// TIA Portal V17 export
// export: Created 2024-06-25T12:57:18.7892853Z, ExportSetting WithDefaults, DisplayName Totally Integrated Automation Portal, DisplayVersion V17 Update 6, DisplayName TIA Portal Openness, DisplayVersion V17 Update 6, DisplayName TIA Portal Version Control Interface, DisplayVersion V17, DisplayName STEP 7 Professional, DisplayVersion V17 Update 6, DisplayName STEP 7 Safety, DisplayVersion V17 Update 6, DisplayName WinCC Advanced, DisplayVersion V17 Update 6
FUNCTION "Salidas" : Void   // FC5, LAD
{ S7_Optimized_Access := 'TRUE' }
VERSION : 0.1
// stored: AutoNumber true, IsIECCheckEnabled false, SetENOAutomatically false, UDAEnableTagReadback false
BEGIN

REGION Network 1: PILOTO OFF
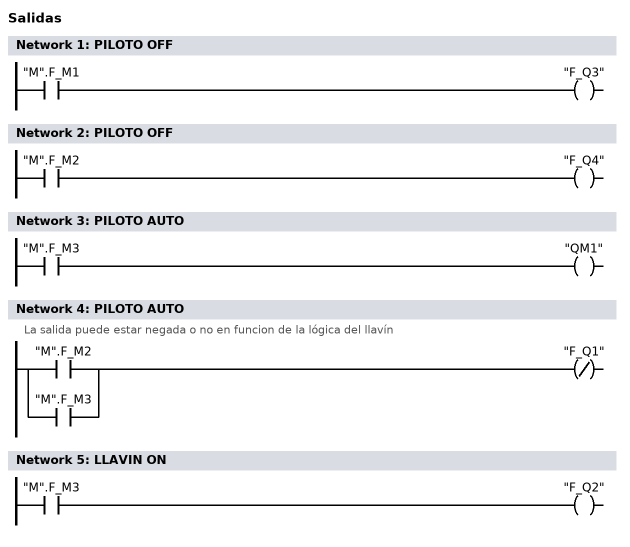
   RUNG wire#powerrail
      Contact( "M".F_M1 )
      Coil( "F_Q3" )
   END_RUNG
   // the same network as SCL:
   "F_Q3" := "M".F_M1;
END_REGION

REGION Network 2: PILOTO OFF
   RUNG wire#powerrail
      Contact( "M".F_M2 )
      Coil( "F_Q4" )
   END_RUNG
   // the same network as SCL:
   "F_Q4" := "M".F_M2;
END_REGION

REGION Network 3: PILOTO AUTO
   RUNG wire#powerrail
      Contact( "M".F_M3 )
      Coil( "QM1" )
   END_RUNG
   // the same network as SCL:
   "QM1" := "M".F_M3;
END_REGION

REGION Network 4: PILOTO AUTO
   // La salida puede estar negada o no en funcion de la lógica del llavín
   RUNG wire#powerrail
      Contact( "M".F_M2 )
      wire#w1
      I_Coil( "F_Q1" )
   END_RUNG
   RUNG wire#powerrail
      Contact( "M".F_M3 )
   END_RUNG wire#w1
   // the same network as SCL:
   "F_Q1" := NOT ("M".F_M2 OR "M".F_M3);
END_REGION

REGION Network 5: LLAVIN ON
   RUNG wire#powerrail
      Contact( "M".F_M3 )
      Coil( "F_Q2" )
   END_RUNG
   // the same network as SCL:
   "F_Q2" := "M".F_M3;
END_REGION
END_FUNCTION
